// TIA Portal V16 export
// export: Created 2020-09-25T08:11:30.4862884Z, ExportSetting WithDefaults, DisplayName Totally Integrated Automation Portal, DisplayVersion V16 Update 2, DisplayName TIA Portal Version Control Interface, DisplayVersion V16 Update 2, DisplayName TIA Portal Openness, DisplayVersion V16 Update 2, DisplayName STEP 7 Professional, DisplayVersion V16 Update 2, DisplayName STEP 7 Safety, DisplayVersion V16, DisplayName WinCC Advanced, DisplayVersion V16 Update 2
FUNCTION_BLOCK "Baustein_2"   // FB2, STL
VERSION : 0.1
// stored: AutoNumber true, UDAEnableTagReadback false
   VAR_INPUT
      input1 : Bool;
      input2 : Bool;
   END_VAR
BEGIN

NETWORK
TITLE = 
      A     #input2;
      A     #input1;
      =     "bool2";



END_FUNCTION_BLOCK
